// TIA Portal project "LAP_2010_2_Transportwagen" (V14)

(* hardware
DEVICE "S7-1200-Station_1"  S7-1200 Station
   slot 0: "Baugruppenträger_0"  S7-1200 Rack  Rack  V1.0
   slot 1: "PLC_1"  CPU 1214C DC/DC/DC  6ES7 214-1AG40-0XB0  V4.2
   slot 3: "AQ 1x12BIT_1"  AQ1 signal board  6ES7 232-4HA30-0XB0  V1.0
*)

// ===== PLC "PLC_1"  CPU 1214C DC/DC/DC =====

VAR_GLOBAL   // PLC tag table "Standard-Variablentabelle"
   "System_Byte" AT %MB100 : Byte;
   "FirstScan" AT %M100.0 : Bool;
   "DiagStatusUpdate" AT %M100.1 : Bool;
   "AlwaysTRUE" AT %M100.2 : Bool;
   "AlwaysFALSE" AT %M100.3 : Bool;
   "Clock_Byte" AT %MB110 : Byte;
   "Clock_10Hz" AT %M110.0 : Bool;
   "Clock_5Hz" AT %M110.1 : Bool;
   "Clock_2.5Hz" AT %M110.2 : Bool;
   "Clock_2Hz" AT %M110.3 : Bool;
   "Clock_1.25Hz" AT %M110.4 : Bool;
   "Clock_1Hz" AT %M110.5 : Bool;
   "Clock_0.625Hz" AT %M110.6 : Bool;
   "Clock_0.5Hz" AT %M110.7 : Bool;
END_VAR

DATA_BLOCK "VersionInput"   // DB1
{ S7_Optimized_Access := 'FALSE' }
VERSION : 0.1
   VAR
      AutoTest : Bool;
      "Version" : String := 'LAP 2010/2 Transportwagen V2.0';
   END_VAR
BEGIN
END_DATA_BLOCK

DATA_BLOCK "DigInput"   // DB2
{ S7_Optimized_Access := 'FALSE' }
VERSION : 0.1
   VAR
      B1 : Bool;   // Endschalter Links
      B2 : Bool;   // Endschalter Rechts
      F1 : Bool;   // Thermorelais
      S1 : Bool;   // Taster Start
      S2 : Bool;   // NotHalt
      S3 : Bool;   // Taster Reset
   END_VAR
BEGIN
END_DATA_BLOCK

DATA_BLOCK "DigOutput"   // DB3
{ S7_Optimized_Access := 'FALSE' }
VERSION : 0.1
   VAR
      P1 : Bool;   // Meldeleuchte Störung
      Q1 : Bool;   // Motor LL
      Q2 : Bool;   // Motor RL
   END_VAR
BEGIN
END_DATA_BLOCK

FUNCTION "DeleteMe" : Void   // FC1, SCL
{ S7_Optimized_Access := 'TRUE' }
VERSION : 0.1
BEGIN
END_FUNCTION

FUNCTION "DatenRangieren" : Void   // FC2, SCL
{ S7_Optimized_Access := 'TRUE' }
VERSION : 0.1
   VAR_TEMP
      ErstesByte : Byte;
      ZweitesByte : Byte;
   END_VAR
BEGIN
   IF "VersionInput".AutoTest THEN
       ; //  Es werden nur die Datenbausteine verwendet  
   ELSE
       // Digitale Eingänge I0.0 - I1.7 in den Datenbaustein DigInput DB2 kopieren
       // IB0 --> DB2 Byte 0
       // IB1 --> DB2 Byte 1
       // Area 16#81 --> Input
       // Area 16#82 --> Output
       // Area 16#84 --> DB
       #ErstesByte := PEEK(area := 16#81, dbNumber := 0, byteOffset := 0);
       #ZweitesByte := PEEK(area := 16#81, dbNumber := 0, byteOffset := 1);

       POKE(area := 16#84,
            dbNumber := 2,
            byteOffset := 0,
            value := #ErstesByte);
       POKE(area := 16#84,
            dbNumber := 2,
            byteOffset := 1,
            value := #ZweitesByte);

       // DB DigOutput auf die Ausgänge Q0.0 - Q1.7 kopieren
       // DB3 Byte 0 --> QB0
       // DB3 Byte 1 --> QB1
       #ErstesByte := PEEK(area := 16#84, dbNumber := 3, byteOffset := 0);
       #ZweitesByte := PEEK(area := 16#84, dbNumber := 3, byteOffset := 1);

       POKE(area := 16#82,
            dbNumber := 0,
            byteOffset := 0,
            value := #ErstesByte);
       POKE(area := 16#82,
            dbNumber := 0,
            byteOffset := 1,
            value := #ZweitesByte);
   END_IF;
END_FUNCTION

ORGANIZATION_BLOCK "Main"   // OB1, LAD, ProgramCycle
TITLE = "Main Program Sweep (Cycle)"
{ S7_Optimized_Access := 'TRUE' }
VERSION : 0.1
   VAR_INPUT
      Initial_Call : Bool;   // Initial call of this OB
      Remanence : Bool;   // =True, if remanent data are available
   END_VAR
BEGIN

REGION Network 1
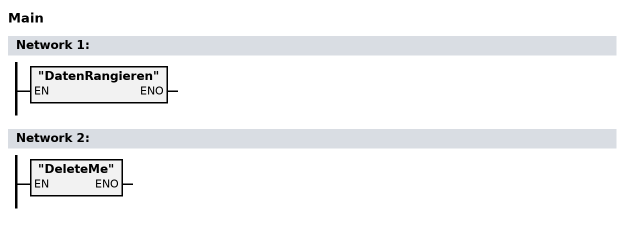
   RUNG wire#powerrail
      "DatenRangieren"()
   END_RUNG
   // the same network as SCL:
   "DatenRangieren"();
END_REGION

REGION Network 2
   RUNG wire#powerrail
      "DeleteMe"()
   END_RUNG
   // the same network as SCL:
   "DeleteMe"();
END_REGION
END_ORGANIZATION_BLOCK

ORGANIZATION_BLOCK "Startup"   // OB100, SCL, Startup
TITLE = "Complete Restart"
{ S7_Optimized_Access := 'TRUE' }
VERSION : 0.1
   VAR_INPUT
      LostRetentive : Bool;   // True if retentive data are lost
      LostRTC : Bool;   // True if date and time are lost
   END_VAR
BEGIN
   "VersionInput".AutoTest := TRUE;

   POKE(area := 16#84,     // DB
        dbNumber := 3,     // DigOutput
        byteOffset := 0,   // Byte 0
        value := byte#0);  // löschen

   POKE(area := 16#84,     // DB
        dbNumber := 3,     // Digoutput
        byteOffset := 1,   // Byte 1
        value := byte#0);  // löschen
END_ORGANIZATION_BLOCK